// TIA Portal project "Contadores" (V16)

(* hardware
DEVICE "S7-1200 station_1"  S7-1200 Station
   slot 0: "Rack_0"  S7-1200 Rack  Rack  V1.0
   slot 1: "PLC_1"  CPU 1214C AC/DC/Rly  6ES7 214-1BG40-0XB0  V4.2
   slot 3: "AQ 1x12BIT_1"  AQ1 signal board  6ES7 232-4HA30-0XB0  V1.0
*)

// ===== PLC "PLC_1"  CPU 1214C AC/DC/Rly =====

VAR_GLOBAL   // PLC tag table "Tabla de variables estándar"
   "Tag_1" AT %MW0 : Int;
   "Tag_2" AT %MW1 : Int;
   "Tag_3" AT %MW3 : Int;
END_VAR

VAR_GLOBAL   // PLC tag table "Marcas"
   "SalidaA_Cont" AT %M0.0 : Bool;
   "SalidaD_Cont" AT %M0.1 : Bool;
   "Valor_Cont" AT %M0.2 : Bool;
   "Personas_recinto" AT %MW2 : Int;
   "FlancoA" AT %M1.0 : Bool;
   "FlancoB" AT %M1.1 : Bool;
   "fotocelulaA_aux" AT %M4.0 : Bool;
   "fotocelulaB_aux" AT %M5.0 : Bool;
END_VAR

VAR_GLOBAL   // PLC tag table "Entradas"
   "Incrementar" AT %I0.0 : Bool;
   "Reset_Cont" AT %I0.1 : Bool;
   "Decrementar" AT %I0.2 : Bool;
   "Cargar_Cont" AT %I0.3 : Bool;
   "fotocelula_A" AT %I0.4 : Bool;
   "fotocelula_B" AT %I0.5 : Bool;
   "Reset_Cont_Recinto" AT %I1.0 : Bool;
   "Carga_Cont_Recinto" AT %I1.1 : Bool;
END_VAR

VAR_GLOBAL   // PLC tag table "Salidas"
   "Lleno" AT %Q0.4 : Bool;
   "Vacio" AT %Q0.5 : Bool;
END_VAR

// folder: System blocks/Program resources

DATA_BLOCK "Cont1"   // DB1
{ S7_Optimized_Access := 'TRUE' }
AUTHOR : Simatic
FAMILY : IEC
NAME : CNTR
VERSION : 1.0
// stored: InstanceOfName IEC_COUNTER
"IEC_COUNTER"
BEGIN
END_DATA_BLOCK

DATA_BLOCK "Cont2"   // DB2
{ S7_Optimized_Access := 'TRUE' }
AUTHOR : Simatic
FAMILY : IEC
NAME : CNTR
VERSION : 1.0
// stored: InstanceOfName IEC_COUNTER
"IEC_COUNTER"
BEGIN
END_DATA_BLOCK

DATA_BLOCK "Cont3"   // DB3
{ S7_Optimized_Access := 'TRUE' }
AUTHOR : Simatic
FAMILY : IEC
NAME : CNTR
VERSION : 1.0
// stored: InstanceOfName IEC_COUNTER
"IEC_COUNTER"
BEGIN
END_DATA_BLOCK

DATA_BLOCK "ContPersonas"   // DB4
{ S7_Optimized_Access := 'TRUE' }
AUTHOR : Simatic
FAMILY : IEC
NAME : CNTR
VERSION : 1.0
// stored: InstanceOfName IEC_COUNTER
"IEC_COUNTER"
BEGIN
END_DATA_BLOCK

// folder: (top level)

ORGANIZATION_BLOCK "Main"   // OB1, LAD, ProgramCycle
TITLE = "Main Program Sweep (Cycle)"
{ S7_Optimized_Access := 'TRUE' }
VERSION : 0.1
   VAR_INPUT
      Initial_Call : Bool;   // Initial call of this OB
      Remanence : Bool;   // =True, if remanent data are available
   END_VAR
   VAR_TEMP   // added for the SCL form of the ladder/FBD networks
      _w1 : Bool;
      _w2 : Bool;
   END_VAR
BEGIN

REGION Network 1: CTU
   // Contador ascendente
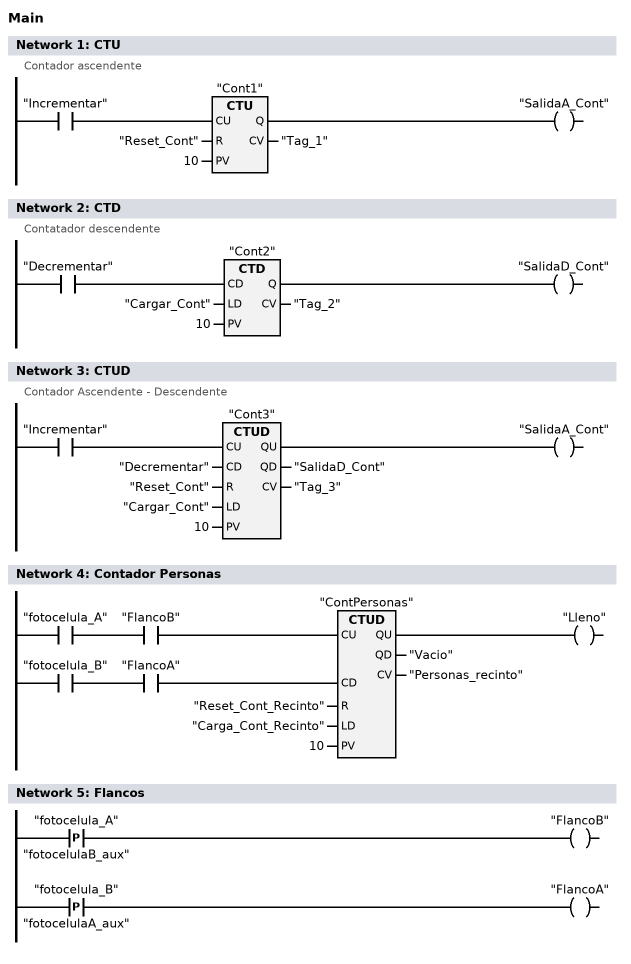
   "Cont1".CTU(CU := "Incrementar", R := "Reset_Cont", PV := 10, CV => "Tag_1");
   "SalidaA_Cont" := "Cont1".Q;
END_REGION

REGION Network 2: CTD
   // Contatador descendente
   "Cont2".CTD(CD := "Decrementar", LD := "Cargar_Cont", PV := 10, CV => "Tag_2");
   "SalidaD_Cont" := "Cont2".Q;
END_REGION

REGION Network 3: CTUD
   // Contador Ascendente ‐ Descendente
   "Cont3".CTUD(CU := "Incrementar",
                CD := "Decrementar",
                R := "Reset_Cont",
                LD := "Cargar_Cont",
                PV := 10,
                QD => "SalidaD_Cont",
                CV => "Tag_3");
   "SalidaA_Cont" := "Cont3".QU;
END_REGION

REGION Network 4: Contador Personas
   "ContPersonas".CTUD(CU := "fotocelula_A" AND "FlancoB",
                       CD := "fotocelula_B" AND "FlancoA",
                       R := "Reset_Cont_Recinto",
                       LD := "Carga_Cont_Recinto",
                       PV := 10,
                       QD => "Vacio",
                       CV => "Personas_recinto");
   "Lleno" := "ContPersonas".QU;
END_REGION

REGION Network 5: Flancos
   RUNG wire#powerrail
      P_Contact(operand := "fotocelula_A", bit := "fotocelulaB_aux")
      Coil( "FlancoB" )
   END_RUNG
   RUNG wire#powerrail
      P_Contact(operand := "fotocelula_B", bit := "fotocelulaA_aux")
      Coil( "FlancoA" )
   END_RUNG
   // the same network as SCL:
   #_w1 := "fotocelula_A" AND NOT "fotocelulaB_aux";   // rising edge of "fotocelula_A"
   "fotocelulaB_aux" := "fotocelula_A";
   "FlancoB" := #_w1;
   #_w2 := "fotocelula_B" AND NOT "fotocelulaA_aux";   // rising edge of "fotocelula_B"
   "fotocelulaA_aux" := "fotocelula_B";
   "FlancoA" := #_w2;
END_REGION
END_ORGANIZATION_BLOCK